FUNCTION_BLOCK LevelControl
VAR_INPUT
	bStart : BOOL;
	bStop : BOOL;
	bReset : BOOL;
	
	rWaterLevel : REAL;
END_VAR
VAR_OUTPUT
	bHighLevel : BOOL;
	bLowLevel : BOOL;
	
	bSolenoidA : BOOL;
	bSolenoidB : BOOL;
	
	bPump : BOOL;
	bAgitator : BOOL;
	
	rPumpPos : LREAL;
	rAgitatorPos : LREAL;
END_VAR
VAR
	iState : UDINT;
	bInitialActivate : BOOL;
	
	fbInitial : R_TRIG;
	
	Agitator : AXIS_REF;
	Pump : AXIS_REF;
	JogAgitator : MC_Jog;
	JogPump : MC_Jog;
	PowerAgitator : MC_Power;
	PowerPump : MC_Power;
END_VAR

bInitialActivate := TRUE; 
fbInitial(CLK := TRUE);
IF fbInitial.Q THEN
	rWaterLevel := 0.0; //sets the starting point for level to 0
END_IF
IF bStart THEN
	JogAgitator(Axis := Agitator,JogForward := TRUE);
END_IF
IF bStop THEN
	JogAgitator(Axis := Agitator,JogForward := FALSE);
END_IF

IF JogPump.Active THEN
	bPump := TRUE;
ELSIF NOT JogPump.Active THEN
	bPump := FALSE;	
END_IF

IF JogAgitator.Active THEN
	bAgitator := TRUE;
ELSIF NOT JogAgitator.Active THEN
	bAgitator := FALSE;	
END_IF

CASE iState OF
	0:
		IF PowerAgitator.Status AND PowerPump.Status THEN
			iState := 10;
		END_IF
	5: //if agitator is turned off reset
		JogPump(Axis := Pump,JogForward := FALSE);
		bSolenoidA := FALSE;
		bSolenoidB := FALSE;
		iState := 0;	
	10://check the water level
		IF JogAgitator.Active THEN
			IF rWaterLevel >= 9.5 AND rWaterLevel < 24.5 THEN
				iState := 20;
			ELSIF rWaterLevel >= 24.5	AND rWaterLevel < 89.5 THEN
				iState := 30;
			ELSIF rWaterLevel < 9.5 AND rWaterLevel > 0.0 THEN
				iState := 40;
			ELSIF rWaterLevel >= 89.5 THEN
				iState := 50;
			END_IF
		END_IF
	20: //fill the reservoir
		IF JogAgitator.Active THEN
			bSolenoidA := TRUE;
			bSolenoidB := TRUE;
			JogPump(Axis := Pump,JogForward := FALSE);
			bHighLevel := FALSE;
			bLowLevel := FALSE;
			iState := 0;
		ELSE
			iState := 5;	
		END_IF
	30: //empty the reservoir
		IF JogAgitator.Active THEN
			JogPump(Axis := Pump,JogForward := TRUE);
			bSolenoidA := FALSE;
			bSolenoidB := FALSE;
			bHighLevel := FALSE;
			bLowLevel := FALSE;
			iState := 0;
		ELSE
			iState := 5;	
		END_IF
	40: //crtitically low level
		IF JogAgitator.Active THEN
			bSolenoidA := FALSE;
			bSolenoidB := FALSE;
			JogPump(Axis := Pump,JogForward := FALSE);
			bHighLevel := FALSE;
			bLowLevel := TRUE;
			IF bReset  THEN
				iState := 100;
			END_IF
		ELSE
			iState := 5;	
		END_IF
	50: //critically high level	
		IF JogAgitator.Active THEN
			bSolenoidA := FALSE;
			bSolenoidB := FALSE;
			JogPump(Axis := Pump,JogForward := FALSE);
			bHighLevel := TRUE;
			bLowLevel := FALSE;
			IF bReset  THEN
				iState := 100;
			END_IF
		ELSE
			iState := 5;	
		END_IF
	100://reset
		bLowLevel := FALSE;
		bHighLevel := FALSE;
		iState := 0;
			 		
END_CASE

PowerAgitator(Axis := Agitator,Enable := TRUE,Enable_Positive := TRUE,Enable_Negative := TRUE);
PowerPump(Axis := Pump,Enable := TRUE,Enable_Positive := TRUE,Enable_Negative := TRUE);

JogAgitator(Axis := Agitator);
JogPump(Axis := Pump);

rPumpPos := Pump.NcToPlc.ActPos;
rAgitatorPos := Agitator.NcToPlc.ActPos;

END_FUNCTION_BLOCK

(* stored: Version 1.1.0.1, ProductVersion 3.1.4024.12
   POU LevelControl: Id {33c21ed2-92f4-474f-9fe3-f60756b7bd1f}, SpecialFunc None *)
